// TIA Portal V19 export
FUNCTION "FC_DP_Error" : Void   // FC203, STL
TITLE = Profibusfehler melden
{ S7_Optimized_Access := 'FALSE' }
// stored: AutoNumber false
   VAR_TEMP
      RetVal : Int;
      Adresse : DWord;
      Count : Int;
      Wert_akt : Byte;
      Wert_alt : Byte;
      Err_Nr : USInt;
      Inf : Struct
         Inf1 : Byte;
         inf2 : Byte;
      END_STRUCT;
   END_VAR
BEGIN

NETWORK
TITLE = Störung/Ausfall
      AN    "DB_ANLAGE".config.Check_Profibus;  //keine Überwachung gefordert
      ON    "DB_ANLAGE".IN.Watch_Profibus;  //Überwachung nicht möglich
      BEC;
      R     "DB_DP_Error".Sammelwarnung;
      R     "DB_DP_Error".Sammelstoerung;

      A     "DB_ANLAGE".IN.PC_offline;  //kein PC-aktiv --> keine Überwachung
      BEC;

//Erstmalige Prüfung?
      AN    "DB_DP_Error".Init;
      AN    "DB_ANLAGE".IN.AMS_Restart;
      JC    norm;


NETWORK
TITLE = erstmalige Prüfung --> nur Fehlerstatus 2oder 3 senden
// Statuswert Bedeutung:
// 0: nicht projektiert & nicht vorhanden
// 1: vorhanden & ok
// 2: vorhanden aber nicht ok
// 3: projektiert aber nicht vorhanden
      SET;
      R     "DB_DP_Error".Init;

//aktuellen Status als Altstatus übernehmen
      CALL  FILL
      ( BVAL    := "DB_DP_Error".DP_Slave,
        RET_VAL := #RetVal,
        BLK     := "DB_DP_Error".Altwert
      );

//Altwert-Einträge mit Status 0,1 bleiben
//Einträge mit 2,3 werden auf 1 gesetzt
//dadurch wird bei fehlerhaften Einträgen ein Wechsel von 1 auf 2 oder 3 erkannt
//und somit erneut gemeldet
      L     0;
      L     "DB_DP_Error".HiAdr;
      ==I;
      BEC;
retC: T     #Count;
      L     1024;
      +D;
      SLD   3;
      T     #Adresse;
      OPN   "DB_DP_Error";
      L     DBB [#Adresse];
      L     1;  //Wert 0,1 bleibt erhalten
      <=I;
      JC    nexC;
      T     DBB [#Adresse];
nexC: L     #Count;
      LOOP  retC;  //Wert 2,3 mit 1 überschreiben

NETWORK
TITLE = Normalprüfung --> jede Statusänderung melden
norm: NOP   0;

      L     0;  //keine Profibusteilnehmer
      L     "DB_DP_Error".HiAdr;
      ==I;
      BEC;
reC:  T     #Count;
      SLD   3;
      T     #Adresse;
      OPN   "DB_DP_Error";
      L     DBB [#Adresse];
      T     #Wert_akt;  //"DB_DP_Error".DP_Slave[#Count]

      L     #Wert_akt;  //Warnung melden
      L     2;
      ==I;
      S     "DB_DP_Error".Sammelwarnung;
      L     #Wert_akt;  //Störung melden
      L     3;
      ==I;
      S     "DB_DP_Error".Sammelstoerung;

      L     #Count;
      +     1024;
      SLD   3;
      T     #Adresse;
      OPN   "DB_DP_Error";
      L     DBB [#Adresse];
      T     #Wert_alt;

//Statusauswertung und Änderung melden
      L     #Wert_akt;  //"DB_DP_Error".Altwert[#Count]
      L     #Wert_alt;
      ==I;
      JC    nxC;
      L     #Wert_alt;
      JL    list;
      JU    old0;
      JU    old1;
      JU    old2;
      JU    old3;
list: JU    nxC;

//Baugruppe war weder projektiert noch vorhanden
old0: L     #Wert_akt;
      T     #Err_Nr;
      JC    evt;

//Baugruppe war projektiert und vorhanden
old1: L     0;  //Wechsel auf 0 ist ok
      L     #Wert_akt;
      ==I;
      JC    nxC;
      T     #Err_Nr;
      JC    evt;

//Baugruppe war projektiert,vorhanden aber fehlerhaft
old2: L     0;  //Wechsel auf 0 ist ok
      L     #Wert_akt;
      ==I;
      JC    nxC;
      T     #Err_Nr;
      JC    evt;

//Baugruppe war projektiert aber nicht vorhanden
old3: L     0;  //Wechsel auf 0 ist ok
      L     #Wert_akt;
      ==I;
      JC    nxC;
      T     #Err_Nr;
      JC    evt;

evt:  NOP   0;
//Err_Nr 1:Station wiederkehr
//Err_Nr 2:Station nicht ok
//Err_Nr 3:Station Ausfall
      CALL  BLKMOV
      ( SRCBLK  := #Count,
        RET_VAL := #RetVal,
        DSTBLK  := #Inf
      );


      L     #Err_Nr;
      L     3;
      ==I;
      A     "DB_DP_Error".Hupe_enable;
      R     "DB_ANLAGE".config.M_Q_Hupe;

nxC:  L     #Count;
      LOOP  reC;

//aktuellen Status als Altstatus übernehmen
      CALL  FILL
      ( BVAL    := "DB_DP_Error".DP_Slave,
        RET_VAL := #RetVal,
        BLK     := "DB_DP_Error".Altwert
      );

END_FUNCTION
